TYPE DUT_ActPos :
STRUCT
		Mode :UINT:=1;
		Pos:REAL:=1.0;
		
END_STRUCT
END_TYPE

(* stored: Version 1.1.0.1, ProductVersion 3.1.4024.9
   DUT DUT_ActPos: Id {712e0482-2f1f-4109-ba39-4b35cefd60ca} *)
